(*********************************** G.D S.p.A. - Technical Department ***********************************
============= PROGRAM INFO ============
FOLDER:             TBD
MACHINES INVOLVED:  TBD 

============= DESCRIPTION =============
csp machine declaration

============= REVISIONS ===============
Date		Version	 	Author      	Description             
----------	-------		------------  	--------------------------------------------
2019/04/05 	0000.00	 	M.Grasso		Creation of the PRG

**********************************************************************************************************)
(*$R process_ref := prc; $*)
PROGRAM csp_case_transport_os
VAR
	
	prc:											process;
	prc_path:										STRING;
	
END_VAR

_read_var_input();

_object_manager();

IF NOT objects_running()
THEN
	RETURN;	
END_IF

_read_process_image();

_mode_manager();

_set_runtime_properties();

(********************************* BODY *********************************)
(************************************************************************)

_handle_messages();

_write_output();

ACTION _handle_messages:
;
END_ACTION

ACTION _handle_process_test:
;
END_ACTION

ACTION _mode_manager:
IF process_mode_req_is_pending(prc)
THEN
    process_apply_mode_req_first_step(prc);
    CASE process_get_mode(prc) OF
        MODE_TO_ABSENT:
			;
        MODE_TO_INACTIVE:
			;
        MODE_TO_TEST:
			;
        MODE_TO_OPERATIONAL:
			;
    END_CASE
    process_apply_mode_req_second_step(prc);
END_IF
END_ACTION

ACTION _object_manager:
IF objects_initialization()
THEN
	sub_process_init(
		object_name					:= 'csp_case_transport_os.prc', 
		process						:= csp_case_transport.prc, 
		CONVERSION_this				:= prc);
		
	prc_path 						:= process_get_path(prc);
END_IF

IF objects_running()
THEN
	process_cycle(prc);
END_IF
END_ACTION

ACTION _read_process_image:
;
END_ACTION

ACTION _read_var_input:
;
END_ACTION

ACTION _set_runtime_properties:
;
END_ACTION

ACTION _write_output:
;
END_ACTION

END_PROGRAM

(* stored: Version 1.1.0.1, ProductVersion 3.1.4022.12
   POU csp_case_transport_os: Id {bc086295-7397-476c-a120-843753aa2864}, SpecialFunc None
   Action _handle_messages: Id {b2fac2ac-d6b0-46ea-a91f-d7bf61e2c449}
   Action _handle_process_test: Id {e679ca3e-0256-4a4f-918f-748aa1672089}
   Action _mode_manager: Id {1ccf6f97-4b5b-46e6-8c2d-c0c57e2599b7}
   Action _object_manager: Id {a945992d-90cf-4643-9bdb-bb0b149068d9}
   Action _read_process_image: Id {38fa664e-a69e-4b04-8969-7f3f57a2b879}
   Action _read_var_input: Id {21eea165-02fe-470d-ac0c-469530650fdf}
   Action _set_runtime_properties: Id {701e422d-5661-4b26-a345-36cd62b300e9}
   Action _write_output: Id {c6eb527d-655b-455f-ae9e-cccbce153fe7} *)
